// SIMATIC STEP 7 (V5.x) project BTL VXL
// CPU: CPU 314C-2 PN/DP
// station: Hardware
// station: SIMATIC 300(1)
// station: P_ADR_BUS
// program: S7 Program(1)

SYMBOL_TABLE
"ON"	I 0.0	BOOL
"OFF"	I 0.1	BOOL
"Gia tri nhiet do"	MD 18	DWORD
"Gia tri so dau vao"	PIW 800	WORD
"Run"	Q 0.0	BOOL
"LA1"	Q 0.1	BOOL
"HA1"	Q 0.2	BOOL
END_SYMBOL_TABLE

ORGANIZATION_BLOCK OB 1
TITLE = "Main Program Sweep (Cycle)"
VERSION : 0.1
VAR_TEMP
  OB1_EV_CLASS : BYTE ;	//Bits 0-3 = 1 (Coming event), Bits 4-7 = 1 (Event class 1)
  OB1_SCAN_1 : BYTE ;	//1 (Cold restart scan 1 of OB 1), 3 (Scan 2-n of OB 1)
  OB1_PRIORITY : BYTE ;	//Priority of OB Execution
  OB1_OB_NUMBR : BYTE ;	//1 (Organization block 1, OB1)
  OB1_RESERVED_1 : BYTE ;	//Reserved for system
  OB1_RESERVED_2 : BYTE ;	//Reserved for system
  OB1_PREV_CYCLE : INT ;	//Cycle time of previous OB1 scan (milliseconds)
  OB1_MIN_CYCLE : INT ;	//Minimum cycle time of OB1 (milliseconds)
  OB1_MAX_CYCLE : INT ;	//Maximum cycle time of OB1 (milliseconds)
  OB1_DATE_TIME : DATE_AND_TIME ;	//Date and time OB1 started
END_VAR
BEGIN
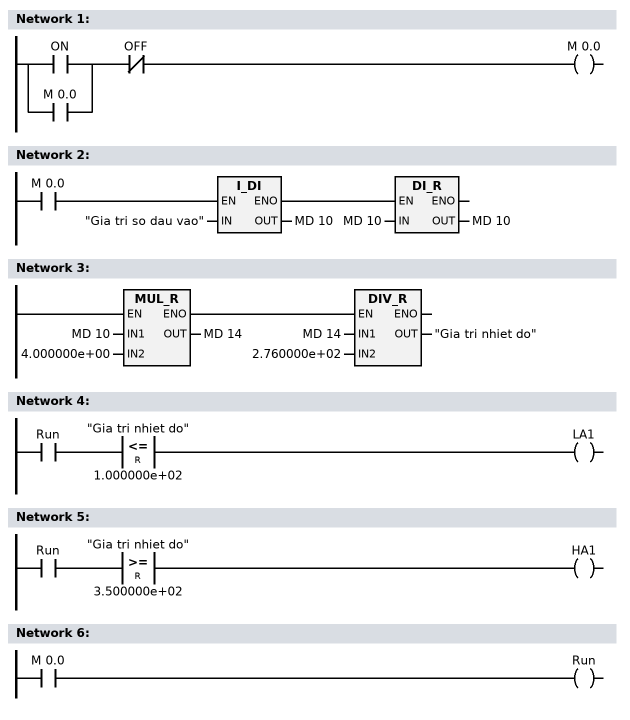
NETWORK
TITLE =
      A(;
      O     "ON";
      O     M 0.0;
      );
      AN    "OFF";
      =     M 0.0;
NETWORK
TITLE =
      A(;
      A     M 0.0;
      JNB   _001;
      L     "Gia tri so dau vao";
      ITD;
      T     MD 10;
      SET;
      SAVE;
      CLR;
_001: A     BR;
      );
      JNB   _002;
      L     MD 10;
      DTR;
      T     MD 10;
_002: NOP   0;
NETWORK
TITLE =
      A(;
      L     MD 10;
      L     4.000000e+00;
      *R;
      T     MD 14;
      AN    OV;
      SAVE;
      CLR;
      A     BR;
      );
      JNB   _003;
      L     MD 14;
      L     2.760000e+02;
      /R;
      T     "Gia tri nhiet do";
_003: NOP   0;
NETWORK
TITLE =
      A     "Run";
      A(;
      L     "Gia tri nhiet do";
      L     1.000000e+02;
      <=R;
      );
      =     "LA1";
NETWORK
TITLE =
      A     "Run";
      A(;
      L     "Gia tri nhiet do";
      L     3.500000e+02;
      >=R;
      );
      =     "HA1";
NETWORK
TITLE =
      A     M 0.0;
      =     "Run";
END_ORGANIZATION_BLOCK
